(* IEC 61131-3 sources: CodesysTest/alpha/export/FBs/DataHandlers/FB_ModbusDWORD.pou/RawValue.prop, 1 file *)

(* ---- Get.pm.st ---- *)
(*#-#-#-#-#-#-#-#-#-#---Declaration---#-#-#-#-#-#-#-#-#-#-#-#-#*)

VAR
END_VAR
(*#-#-#-#-#-#-#-#-#-#---Implementation---#-#-#-#-#-#-#-#-#-#-#-#-#*)

_rawValue := OSCAT_BASIC.DWORD_OF_WORD(_highWord,_lowWord);
RawValue := _rawValue;
